(* IEC 61131-3 sources: inproshop/test7_exported/1.Function/FB/Robot(机械手)/Epson, 4 files *)

(* ---- Str_Epson.st ---- *)
TYPE Str_Epson :
STRUCT
	Cmd:Str_EpsonCmd;//控制
	Status:Str_EpsonStatus;//状态
END_STRUCT
END_TYPE

(* ---- Str_EpsonCmd.st ---- *)
TYPE Str_EpsonCmd :
STRUCT
	Rob_Start		:BOOL;//启动（IN512）
	Rob_Stop		:BOOL;//停止（IN513）
	Rob_Pause		:BOOL;//暂停（IN514）
	Rob_Continue	:BOOL;//继续（IN515）
	Rob_Reset		:BOOL;//复位（IN516）
	SetMotorsOn		:BOOL;//伺服使能打开（IN517）
	SetMotorsOff	:BOOL;//伺服使能关闭（IN518）
	SetPowerHigh	:BOOL;//高功率模式（IN519）
	SetPowerLow		:BOOL;//低功率模式（IN520）
	X_For			:BOOL;//X正向点动（IN521）
	X_Back			:BOOL;//X反向点动（IN522）
	Y_For			:BOOL;//Y正向点动（IN523）
	Y_Back			:BOOL;//Y反向点动（IN524）
	Z_For			:BOOL;//Z正向点动（IN525）
	Z_Back			:BOOL;//Z反向点动（IN526）
	U_For			:BOOL;//U正向点动(IN527)
	U_Back			:BOOL;//U反向点动(IN528)
	V_For			:BOOL;//V正向点动(IN529)
	V_Back			:BOOL;//V反向点动(IN530)
	W_For			:BOOL;//W正向点动(IN531)
	W_Back			:BOOL;//W反向点动(IN532)
	SavePoint		:BOOL;//点位保存(IN533)
	Rob_Jump		:BOOL;//执行JUMP运动(IN534)
	ManuMode		:BOOL;//手动模式(IN535)
	AutoMode		:BOOL;//自动模式(IN536)
	SFree			:BOOL;//电机释放(IN537)
	SLock			:BOOL;//电机锁定(IN538)
	TeachMode		:BOOL;//示教模式(IN539)
	SpaceBoo29		:BOOL;//预备位(IN540)
	MachineIntial	:BOOL;//设备初始化(IN541)
	MachineAutoRun	:BOOL;//设备自动中(IN542)
	MachineStepRun	:BOOL;//单步信号(IN543)
	Speed			:INT;//	运行速度(IN34)
	PointNum		:INT;//	选择点位(IN35)
	InterFace_B:ARRAY[576..607] OF BOOL;//交互信号
	ProductType		:INT;//产品型号(IN38)
	InterFace_IN39	:INT;//交换数据字(IN39)
	InterFace_IN40	:INT;//交换数据字(IN40)
	InterFace_IN41	:INT;//交换数据字(IN41)
	InterFace_IN42	:INT;//交换数据字(IN42)
	InterFace_IN43	:INT;//交换数据字(IN43)
	InterFace_IN44	:INT;//交换数据字(IN44)
	InterFace_IN45	:INT;//交换数据字(IN45)
	InterFace_IN46	:INT;//交换数据字(IN46)
	InterFace_IN47	:INT;//交换数据字(IN47)
	InterFace_IN48	:INT;//交换数据字(IN48)
	InterFace_IN49	:INT;//交换数据字(IN49)
	InterFace_IN50	:INT;//交换数据字(IN50)
	InterFace_IN51	:INT;//交换数据字(IN51)
	InterFace_IN52	:INT;//交换数据字(IN52)
	InterFace_IN53	:INT;//交换数据字(IN53)

END_STRUCT
END_TYPE

(* ---- Str_EpsonStatus.st ---- *)
TYPE Str_EpsonStatus :
STRUCT
	Ready:			BOOL;//	准备好（OUT512）
	Running:		BOOL;//	运转中（OUT513）
	Paused:			BOOL;//	暂停中（OUT514）
	Error:			BOOL;//	错误（OUT515）
	EStopOn:		BOOL;//	急停（OUT516）
	SafeguardOn:	BOOL;//	安全门（OUT517）
	SError:			BOOL;//	重故障（OUT518）
	Warning:		BOOL;//	警告（OUT519）
	MotorsOn:		BOOL;//	伺服使能打开（OUT520）
	AtHome:			BOOL;//	机器人在原点（OUT521）
	PowerHigh:		BOOL;//	高功率模式（OUT522）
	ResetOver:		BOOL;//	主程序编号2（OUT523）
	Free:			BOOL;//	电机已释放（OUT524）
	Lock:			BOOL;//	电机已锁住（OUT525）
	TeachOver:		BOOL;//	示教完成（OUT526）
	Intialed:		BOOL;//	机械手初始化完成(OUT527)
	ErrorCode:		WORD;//	错误代码（OUT528-541）（OUT33）
	InsideBox1:		BOOL;//	Box1（OUT544）
	InsideBox2:		BOOL;//	Box2（OUT545）
	InsideBox3:		BOOL;//	Box3（OUT546）
	InsideBox4:		BOOL;//	Box4（OUT547）
	InsideBox5:		BOOL;//	Box5（OUT548）
	InsideBox6:		BOOL;//	Box6（OUT549）
	InsideBox7:		BOOL;//	Box7（OUT550）
	InsideBox8:		BOOL;//	Box8（OUT551）
	InsideBox9:		BOOL;//	Box9（OUT552）
	InsideBox10:	BOOL;//	Box10（OUT553）
	InsideBox11:	BOOL;//	Box11（OUT554）
	InsideBox12:	BOOL;//	Box12（OUT555）
	InsideBox13:	BOOL;//	Box13（OUT556）
	InsideBox14:	BOOL;//	Box14（OUT557）
	InsideBox15:	BOOL;//	Box15（OUT558）
	Space2:			BOOL;//	预备位
	InsidePlane1:	BOOL;//	Plane1（OUT560）
	InsidePlane2:	BOOL;//	Plane2（OUT561）
	InsidePlane3:	BOOL;//	Plane3（OUT562）
	InsidePlane4:	BOOL;//	Plane4（OUT563）
	InsidePlane5:	BOOL;//	Plane5（OUT564）
	InsidePlane6:	BOOL;//	Plane6（OUT565）
	InsidePlane7:	BOOL;//	Plane7（OUT566）
	InsidePlane8:	BOOL;//	Plane8（OUT567）
	InsidePlane9:	BOOL;//	Plane9（OUT568）
	InsidePlane10:	BOOL;//	Plane10（OUT569）
	InsidePlane11:	BOOL;//	Plane11（OUT570）
	InsidePlane12:	BOOL;//	Plane12（OUT571）
	InsidePlane13:	BOOL;//	Plane13（OUT572）
	InsidePlane14:	BOOL;//Plane14（OUT573）
	InsidePlane15:	BOOL;//	Plane15（OUT574）
	Space3:			BOOL;//	预备位
	InterFace_B:ARRAY[576..607] OF BOOL;//交互信号
	InterFace_OUT38:	WORD;// 交换数据字(OUT38)
	InterFace_OUT39:	WORD;//	交换数据字(OUT39)
	InterFace_OUT40:	WORD;// 交换数据字(OUT40)
	InterFace_OUT41:	WORD;//	交换数据字(OUT41)
	InterFace_OUT42:	WORD;//	交换数据字(OUT42)
	InterFace_OUT43:	WORD;//	交换数据字(OUT43)
	InterFace_OUT44:	WORD;//	交换数据字(OUT44)
	InterFace_OUT45:	WORD;//	交换数据字(OUT45)
	InterFace_OUT46:	WORD;//	交换数据字(OUT46)
	InterFace_OUT47:	WORD;//	交换数据字(OUT47)
END_STRUCT
END_TYPE

(* ---- FB_Epson_V1.st ---- *)
FUNCTION_BLOCK FB_Epson_V1
VAR_IN_OUT
	ioEpson:Str_Epson;
END_VAR
VAR_INPUT
	iMode:Str_Mode;//设备控制模式
	iName:WSTRING;//名称
	iDstAdr:STRING;//IP地址
	iDstTcpPort:UINT;//端口号
	iSpeed:REAL;//运行速度
	iProductType:INT;//配方名称
	iClock:BOOL;//发送时钟
END_VAR
VAR_OUTPUT
	oTimeOut:BOOL;//通讯超时
END_VAR
VAR
	i:INT;//循环变量用
	FB_TcpClient_instance:FB_TcpClient;//通讯功能块实例化
	TcpClient:Str_TcpClient;
	bySendData:ARRAY[0..500]OF BYTE;
	byRevData:ARRAY[0..500]OF BYTE;
	change:BOOL;//切换读写状态
	TimeDelayExcute:TON;//数据发送间隔
	TimeDelayExcute_R:R_TRIG;
	TimeDelayControl:ARRAY[0..9] OF TON;//控制延时
	TimeOutDelay:TON;//超时
	EnableDelay:TON;//延时使能
END_VAR

ACT_Input();
ACT_Control();
ACT_Output();
ACT_Socket();
